PROGRAM Prg_Git
VAR
	bTest				: BOOL;
	nTest				: INT;
	fTest				: real;
END_VAR

IF bTest THEN
	nTest := 3;
	fTest := 3.33333;
END_IF

END_PROGRAM

(* stored: Version 1.1.0.1, ProductVersion 3.1.4024.12
   POU Prg_Git: Id {0047a2f0-fe0b-47ae-b3d6-377bcce04bc2}, SpecialFunc None *)
